// TwinCAT 3 PLC project PLC1
// ProgramVersion: 3.1.4024.12
// libraries:
//   Tc2_MC2, * (Beckhoff Automation GmbH)
//   Tc2_NC, * (Beckhoff Automation GmbH)
//   Tc2_Standard, * (Beckhoff Automation GmbH)
//   Tc2_System, * (Beckhoff Automation GmbH)
//   Tc3_MC2_AdvancedHoming, * (Beckhoff Automation GmbH)
//   Tc3_Module, * (Beckhoff Automation GmbH)
// project tree:
//   DUTs/ E_FT.TcTLEO, E_MoveState.TcDUT
//   GVLs/constants/ GVL_AlarmMessage.TcGVL, GVL_InitialSetting.TcGVL
//   GVLs/ GVL_HMI.TcGVL, GVL_IO.TcGVL, GVL_var.TcGVL
//   / PlcTask.TcTTO
//   POUs/BaseFuntion/ FB_CheckFeedback.TcPOU, FB_SetAlarm.TcPOU, FB_TransmitStatesToHMI.TcPOU
//   POUs/ FB_CasingVibratoryBowl1.TcPOU, FB_CorePress.TcPOU, FB_CoreSwaging.TcPOU, FB_CoreVibratoryBowl2.TcPOU, FB_Motor1.TcPOU, FB_OilPump.TcPOU, MAIN.TcPOU
// real-time tasks:
//   TASK PlcTask: cycle T#10ms, priority 20, ADS port 350
// motion (NC):
//   TASK NC-Task 1 SAF: cycle T#2ms, priority 4, ADS port 501
//   TASK NC-Task 1 SVB: cycle T#10ms, priority 8, ADS port 511
//   AXIS Axis 1 (id 1)
//     OtherSettings: AllowMotionCmdToSlave=true
//     encoder EncType=19
//       EncPara: MaxCount=#xffffffff
//     drive DrvType=16
//       DrvPara: MaxCount=#xffffffff, DriveControlDWord=#x00020000
//         Analog: TorqueSetpointScale=10, ScaleFactorActTorque=0.1
//         TimeComp: TaskDelayCycles=1
//     controller CtrType=1
//       CtrPara: PriorControlFactor=1
//         Observer: BandWidth=20
// I/O:
//   DEVICE Device 5 (EtherCAT), AmsNetId 169.254.43.171.6.1
//     Coupler (EK1100) [EK1100 EtherCAT Coupler (2A E-Bus)]
//       Slot1-DI (EL1809) [EL1809 16Ch. Dig. Input 24V, 3ms]
//       Slot2-DI (EL1809) [EL1809 16Ch. Dig. Input 24V, 3ms]
//       Slot3-DI (EL1809) [EL1809 16Ch. Dig. Input 24V, 3ms]
//       Slot4-AI (EL3072) [EL3072 2Ch. Ana. Input +/-10V, +/-20mA]
//       Slot5-DO (EL2809-0015) [EL2809-0015 16Ch. Dig. Output 24V DC, 0.35A, not short-circuit proof]
//       Slot6-DO (EL2809-0015) [EL2809-0015 16Ch. Dig. Output 24V DC, 0.35A, not short-circuit proof]
//       Slot7-DO (EL2809-0015) [EL2809-0015 16Ch. Dig. Output 24V DC, 0.35A, not short-circuit proof]
//       EndTerminal (EL9011) [EL9011 End Terminal]
//     Drive 9 (IHSS57/60-EC) [IHSS57/60-EC]
// variable links:
//   NC-Task 1 SAF/Axes/Axis 1 <-> Device 5 (EtherCAT)/Drive 9 (IHSS57/60-EC)
//     Drive/Inputs/In/nDcOutputTime <-> InfoData/DcOutputShift
//     Drive/Inputs/In/nState1 <-> TxPdoMapping/statusword
//     Drive/Inputs/In/nState2 <-> TxPdoMapping/statusword @bit 8
//     Drive/Inputs/In/nState4 @bit 1 <-> WcState/InputToggle
//     Drive/Inputs/In/nState4 <-> WcState/WcState
//     Drive/Inputs/In/nState5 <-> TxPdoMapping/op_mode_display
//     Drive/Outputs/Out/nCtrl1 <-> RxPdoMapping/controlword
//     Drive/Outputs/Out/nCtrl2 <-> RxPdoMapping/controlword @bit 8
//     Drive/Outputs/Out/nCtrl5 <-> RxPdoMapping/op_mode
//     Drive/Outputs/Out/nDataOut1 <-> RxPdoMapping/target_position
//     Enc/Inputs/In/nDataIn1 <-> TxPdoMapping/actual_position
//     Enc/Inputs/In/nDataIn3 <-> TxPdoMapping/Touch_probe_pos1_pos_value
//     Enc/Inputs/In/nDataIn5 <-> TxPdoMapping/Touch_probe_pos2_pos_value
//     Enc/Inputs/In/nDataIn4 <-> TxPdoMapping/Touch_probe_pos1_neg_value
//     Enc/Inputs/In/nDataIn6 <-> TxPdoMapping/Touch_probe_pos2_neg_value
//     Enc/Inputs/In/nDcInputTime <-> InfoData/DcInputShift
//     Enc/Inputs/In/nState4 @bit 1 <-> WcState/InputToggle
//     Enc/Inputs/In/nState4 <-> WcState/WcState
//     Enc/Inputs/In/nState5 <-> TxPdoMapping/Touch_probe_status
//     Enc/Inputs/In/nState6 <-> TxPdoMapping/Touch_probe_status @bit 8
//     Enc/Outputs/Out/nCtrl5 <-> RxPdoMapping/Touch_probe_function
//     Enc/Outputs/Out/nCtrl6 <-> RxPdoMapping/Touch_probe_function @bit 8
//   PLC1/PLC1 Instance <-> Device 5 (EtherCAT)/Coupler (EK1100)/Slot1-DI (EL1809)
//     PlcTask Inputs/GVL_IO.DI_24VDC_CB_OK <-> Channel 1/Input
//     PlcTask Inputs/GVL_IO.DI_CYL{1..6}_E <-> Channel {6..16 step 2}/Input  (6 links)
//     PlcTask Inputs/GVL_IO.DI_CYL{1..5}_R <-> Channel {7..15 step 2}/Input  (5 links)
//     PlcTask Inputs/GVL_IO.DI_ESR1 <-> Channel 2/Input
//     PlcTask Inputs/GVL_IO.DI_LS1 <-> Channel 4/Input
//     PlcTask Inputs/GVL_IO.DI_M1 <-> Channel 3/Input
//     PlcTask Inputs/GVL_IO.DI_TS1 <-> Channel 5/Input
//   PLC1/PLC1 Instance <-> Device 5 (EtherCAT)/Coupler (EK1100)/Slot2-DI (EL1809)
//     PlcTask Inputs/GVL_IO.DI_CYL6_R <-> Channel 1/Input
//     PlcTask Inputs/GVL_IO.DI_CYL7_R <-> Channel 3/Input
//     PlcTask Inputs/GVL_IO.DI_CYL7_E <-> Channel 2/Input
//     PlcTask Inputs/GVL_IO.DI_ECS <-> Channel 11/Input
//     PlcTask Inputs/GVL_IO.DI_EPD <-> Channel 12/Input
//     PlcTask Inputs/GVL_IO.DI_JLU <-> Channel 13/Input
//     PlcTask Inputs/GVL_IO.DI_PCYL1_E <-> Channel 7/Input
//     PlcTask Inputs/GVL_IO.DI_PCYL2_E <-> Channel 9/Input
//     PlcTask Inputs/GVL_IO.DI_PCYL1_R <-> Channel 8/Input
//     PlcTask Inputs/GVL_IO.DI_PCYL2_R <-> Channel 10/Input
//     PlcTask Inputs/GVL_IO.DI_PE1 <-> Channel 14/Input
//     PlcTask Inputs/GVL_IO.DI_PE2 <-> Channel 15/Input
//     PlcTask Inputs/GVL_IO.DI_PE3 <-> Channel 16/Input
//     PlcTask Inputs/GVL_IO.DI_PS1 <-> Channel 6/Input
//   PLC1/PLC1 Instance <-> Device 5 (EtherCAT)/Coupler (EK1100)/Slot3-DI (EL1809)
//     PlcTask Inputs/GVL_IO.DI_PE4 <-> Channel 1/Input
//     PlcTask Inputs/GVL_IO.DI_PE5 <-> Channel 2/Input
//     PlcTask Inputs/GVL_IO.DI_PE6 <-> Channel 3/Input
//   PLC1/PLC1 Instance <-> Device 5 (EtherCAT)/Coupler (EK1100)/Slot4-AI (EL3072)
//     PlcTask Inputs/GVL_IO.AI_PT1 <-> AI Standard Channel 1/Value
//     PlcTask Inputs/GVL_IO.AI_PT2 <-> AI Standard Channel 2/Value
//   PLC1/PLC1 Instance <-> Device 5 (EtherCAT)/Coupler (EK1100)/Slot5-DO (EL2809-0015)
//     PlcTask Outputs/GVL_IO.DO_CYL{1..6}_E <-> Channel {6..16 step 2}/Output  (6 links)
//     PlcTask Outputs/GVL_IO.DO_CYL{1..5}_R <-> Channel {7..15 step 2}/Output  (5 links)
//     PlcTask Outputs/GVL_IO.DO_M1 <-> Channel 1/Output
//     PlcTask Outputs/GVL_IO.DO_M2 <-> Channel 2/Output
//     PlcTask Outputs/GVL_IO.DO_SV1 <-> Channel 5/Output
//     PlcTask Outputs/GVL_IO.DO_VB1 <-> Channel 3/Output
//     PlcTask Outputs/GVL_IO.DO_VB2 <-> Channel 4/Output
//   PLC1/PLC1 Instance <-> Device 5 (EtherCAT)/Coupler (EK1100)/Slot6-DO (EL2809-0015)
//     PlcTask Outputs/GVL_IO.DO_CYL6_R <-> Channel 1/Output
//     PlcTask Outputs/GVL_IO.DO_CYL7_R <-> Channel 3/Output
//     PlcTask Outputs/GVL_IO.DO_CYL8_R <-> Channel 5/Output
//     PlcTask Outputs/GVL_IO.DO_CYL7_E <-> Channel 2/Output
//     PlcTask Outputs/GVL_IO.DO_CYL8_E <-> Channel 4/Output
//     PlcTask Outputs/GVL_IO.DO_LGreen <-> Channel 16/Output
//     PlcTask Outputs/GVL_IO.DO_PCYL1_E <-> Channel 6/Output
//     PlcTask Outputs/GVL_IO.DO_PCYL2_E <-> Channel 8/Output
//     PlcTask Outputs/GVL_IO.DO_PCYL3_E <-> Channel 10/Output
//     PlcTask Outputs/GVL_IO.DO_PCYL4_E <-> Channel 11/Output
//     PlcTask Outputs/GVL_IO.DO_PCYL5_E <-> Channel 12/Output
//     PlcTask Outputs/GVL_IO.DO_PCYL6_E <-> Channel 13/Output
//     PlcTask Outputs/GVL_IO.DO_PCYL1_R <-> Channel 7/Output
//     PlcTask Outputs/GVL_IO.DO_PCYL2_R <-> Channel 9/Output
//   PLC1/PLC1 Instance <-> Device 5 (EtherCAT)/Coupler (EK1100)/Slot7-DO (EL2809-0015)
//     PlcTask Outputs/GVL_IO.DO_LRed <-> Channel 1/Output
//   PLC1/PLC1 Instance <-> NC-Task 1 SAF/Axes/Axis 1
//     PlcTask Inputs/GVL_IO.AxisRef1.NcToPlc <-> Outputs/ToPlc
//     PlcTask Outputs/GVL_IO.AxisRef1.PlcToNc <-> Inputs/FromPlc

CONFIGURATION PLC1
    RESOURCE PLC ON TwinCAT3
        TASK PlcTask(INTERVAL := T#10ms, PRIORITY := 20);
        PROGRAM Main WITH PlcTask : Main;
    END_RESOURCE
END_CONFIGURATION

// ---- DUTs/E_FT.TcTLEO
{attribute 'qualified_only'}
{attribute 'strict'}
TYPE E_FT :
(
	PUMP,
	
	CYL1_E,
	CYL1_R,
	CYL2_E,
	CYL2_R,
	CYL3_E,
	CYL3_R,
	CYL4_E,
	CYL4_R,
	CYL5_E,
	CYL5_R,
	CYL6_E,
	CYL6_R,
	CYL7_E,
	CYL7_R,
	
	PCYL1_E,
	PCYL1_R,
	PCYL2_E,
	PCYL2_R
);
END_TYPE

// ---- DUTs/E_MoveState.TcDUT
{attribute 'qualified_only'}
{attribute 'strict'}
TYPE E_MoveState :
(
	init,
	enable,
	forward,
	backwards,
	backwards_slow,
	new_target_position,
	error,
	reset
);
END_TYPE

// ---- GVLs/constants/GVL_AlarmMessage.TcGVL
{attribute $27qualified_only$27}
VAR_GLOBAL CONSTANT
	DC : STRING := '24 DC Power Off!';
	ESR1 : STRING := 'Emergency Stop Relay 1 failed!';
	LS1 : STRING := 'Low Oil Level Sw failed!';
	TS1 : STRING := 'High Oil Temp Sw failed!';
	PS1 : STRING := 'Low Air Pressure Switch failed!';
	
	PUMP : STRING := 'Pump isn$27t started to run!';
	PUMP_OFF : STRING := 'Pump isn$27t stopped To run!';
	
	ECS : STRING := 'Operator interface Enable Core Swaging (Stayput Switch) failed!';
	
	CYL1_NOT_EXTENDED : STRING := 'Cylinder 1 isn$27t be extended!'; 
	CYL1_NOT_EXTENDED_OFF : STRING := 'Cylinder 1 isn$27t be de-extended!'; 
	CYL1_NOT_RETRACTED : STRING := 'Cylinder 1 isn$27t be retracted!'; 
	CYL1_NOT_RETRACTED_OFF : STRING := 'Cylinder 1 isn$27t be de-retracted!'; 
	CYL2_NOT_EXTENDED : STRING := 'Cylinder 2 isn$27t be extended!'; 
	CYL2_NOT_EXTENDED_OFF : STRING := 'Cylinder 2 isn$27t be de-extended!'; 
	CYL2_NOT_RETRACTED : STRING := 'Cylinder 2 isn$27t be retracted!';
	CYL2_NOT_RETRACTED_OFF : STRING := 'Cylinder 2 isn$27t be de-retracted!'; 
	CYL3_NOT_EXTENDED : STRING := 'Cylinder 3 isn$27t be extended!';  
	CYL3_NOT_EXTENDED_OFF : STRING := 'Cylinder 3 isn$27t be de-extended!'; 
	CYL3_NOT_RETRACTED : STRING := 'Cylinder 3 isn$27t be retracted!';
	CYL3_NOT_RETRACTED_OFF : STRING := 'Cylinder 3 isn$27t be de-retracted!'; 
	CYL4_NOT_EXTENDED : STRING := 'Cylinder 4 isn$27t be extended!';  
	CYL4_NOT_EXTENDED_OFF : STRING := 'Cylinder 4 isn$27t be de-extended!'; 
	CYL4_NOT_RETRACTED : STRING := 'Cylinder 4 isn$27t be retracted!';
	CYL4_NOT_RETRACTED_OFF : STRING := 'Cylinder 4 isn$27t be de-retracted!'; 
	CYL5_NOT_EXTENDED : STRING := 'Cylinder 5 isn$27t be extended!'; 
	CYL5_NOT_EXTENDED_OFF : STRING := 'Cylinder 5 isn$27t be de-extended!'; 
	CYL5_NOT_RETRACTED : STRING := 'Cylinder 5 isn$27t be retracted!'; 
	CYL5_NOT_RETRACTED_OFF : STRING := 'Cylinder 5 isn$27t be de-retracted!'; 
	CYL6_NOT_EXTENDED : STRING := 'Cylinder 6 isn$27t extended!'; 
	CYL6_NOT_EXTENDED_OFF : STRING := 'Cylinder 6 isn$27t de-extended!';
	CYL6_NOT_RETRACTED : STRING := 'Cylinder 6 isn$27t be retracted!';
	CYL6_NOT_RETRACTED_OFF : STRING := 'Cylinder 6 isn$27t be de-retracted!'; 
	CYL7_NOT_EXTENDED : STRING := 'Cylinder 7 isn$27t extended!'; 
	CYL7_NOT_EXTENDED_OFF : STRING := 'Cylinder 7 isn$27t de-extended!';
	CYL7_NOT_RETRACTED : STRING := 'Cylinder 7 isn$27t be retracted!';
	CYL7_NOT_RETRACTED_OFF : STRING := 'Cylinder 7 isn$27t be de-retracted!'; 
	
	PCYL1_NOT_EXTENDED : STRING := 'Pneumatic Cylinder 1 isn$27t be extended!';
	PCYL1_NOT_EXTENDED_OFF : STRING := 'Pneumatic Cylinder 1 isn$27t be de-extended!'; 
	PCYL1_NOT_RETRACTED : STRING := 'Pneumatic Cylinder 1 isn$27t be retracted!'; 
	PCYL1_NOT_RETRACTED_OFF : STRING := 'Pneumatic Cylinder 1 isn$27t be de-retracted!'; 
	PCYL2_NOT_EXTENDED : STRING := 'Pneumatic Cylinder 2 isn$27t be extended!'; 
	PCYL2_NOT_EXTENDED_OFF : STRING := 'Pneumatic Cylinder 2 isn$27t be de-extended!';
	PCYL2_NOT_RETRACTED : STRING := 'Pneumatic Cylinder 2 isn$27t be retracted!';
	PCYL2_NOT_RETRACTED_OFF : STRING := 'Pneumatic Cylinder 2 isn$27t be de-retracted!'; 
	
	// Vibratory
	PE1_FAIL : STRING := 'Vibratory Bowl 1 Product In Pos PE1 fail!';
	PE2_FAIL : STRING := 'Vibratory Bowl 1 Product Invert PE2 fail!';
	PE3_FAIL : STRING := 'Vibratory Bowl 2 Product In Pos PE3 fail!';
	PE4_FAIL : STRING := 'Vibratory Bowl 1 Product High Level PE4 fail!';	
	PE5_FAIL : STRING := 'Low Lead Spool!';
	
END_VAR

// ---- GVLs/constants/GVL_InitialSetting.TcGVL
{attribute 'qualified_only'}
VAR_GLOBAL CONSTANT
	PUMP_FeedbackCheckingTime : INT := 2000; // ms
	PUMP_RunningDelayTime : INT := 2000; // ms
	
	CYLINDER_FeedbackCheckingTime : INT := 3000; // ms
	
	PCYLINDER1EXTENDED_RunningTime: INT := 100;
	PCYLINDER1RETRACTED_RunningTime: INT := 100;
	PCYLINDER2EXTENDED_RunningTime: INT := 100;
	CYLINDER1EXTENDED_RunningTime: INT := 100;
	CYLINDER1RETRACTED_RunningTime: INT := 100;
	CYLINDER2EXTENDED_RunningTime: INT := 100;
	CYLINDER2RETRACTED_RunningTime: INT := 100;
	CYLINDER3EXTENDED_RunningTime: INT := 100;
	CYLINDER3RETRACTED_RunningTime: INT := 100;
	CYLINDER4EXTENDED_RunningTime: INT := 100;
	CYLINDER4RETRACTED_RunningTime: INT := 100;
	CYLINDER5EXTENDED_RunningDelayTime: INT := 250;
	CYLINDER5RETRACTED_RunningDelayTime: INT := 50;
	CYLINDER6RETRACTED_RunningDelayTime: INT := 50;
	CYLINDER6EXTENDED_RunningDelayTime: INT := 50;
	CYLINDER7RETRACTED_RunningDelayTime: INT := 50;
	CYLINDER7EXTENDED_RunningDelayTime: INT := 50;
	
	M3_RunningDelayTime : INT := 50;
	BOWL_RunningDelayTime : INT := 50;
	
	// for BOWL1
	PCYLINDER3EXTENDED_RunningTime: INT := 250;
	PE2_CheckingDelayTime: INT := 100;
	PE2_MaintainTime: INT := 10;
	PCYLINDER5EXTENDED_RunningTime: INT := 250;
	PCYLINDER4EXTENDED_RunningTime: INT := 150;
	PE4_MaintainTime: INT := 500;
	VB1_MaintainTime: INT := 50;
	
	// for BOWL2
	PCYLINDER6EXTENDED_RunningTime: INT := 250;
	PE6_MaintainTime: INT := 500;
	VB2_MaintainTime: INT := 50;
	
	PUMP_FAN_DelayTime : INT := 10000;
	PUMP_RestartingTime: INT := 3000;
	
	CASING_COUNT_FOR_STARTING : INT := 5;
	CORE_COUNT_FOR_STARTING : INT := 5;
END_VAR

// ---- GVLs/GVL_HMI.TcGVL
VAR_GLOBAL
	// Manual Control
	bManualControl : BOOL := FALSE;
		// motor1
	MC_M1_bSet : BOOL := FALSE;
	MC_M1_rPos : REAL := 0.0;
	MC_M1_rVel : REAL := 0.0;
	MC_M1_rAcc : REAL := 0.0;
	MC_M1_rDec : REAL := 0.0;	

	// safeties
	i_b24VDC_CB_OK : BOOL := FALSE;
	i_bESR1 : BOOL := FALSE;
	i_bLS1 : BOOL := FALSE;
	i_bTS1 : BOOL := FALSE;
	i_bPS1 : BOOL := FALSE;
	bSafeties :BOOL := TRUE;
	
	// signals from HMI
	i_nCmd_Reset : SINT := 0;	// reset Alarm; 0:NoAction, 1:Act, 2:AcceptToAct
	i_nCmd_ClearCount : SINT := 0;	// clear casing count and core count; 0:NoAction, 1:Act, 2:AcceptToAct
	i_nCmd_ResetSetting : SINT := 0;	// reset setting; 0:NoAction, 1:Act, 2:AcceptToAct
	i_nCmd_ResetAlarm : SINT := 0;	// reset Alarm; 0:NoAction, 1:Act, 2:AcceptToAct
	
		// settings
	i_nCoreSwagingMode: INT := 0;	// 0: Auto, 1: Manual
	i_nCasingCountForStarting : INT := GVL_InitialSetting.CASING_COUNT_FOR_STARTING;
	i_nCoreCountForStarting : INT := GVL_InitialSetting.CORE_COUNT_FOR_STARTING;
	i_nPumpFeedbackCheckingTime : INT := GVL_InitialSetting.PUMP_FeedbackCheckingTime; // ms
	i_nCylinderFeedbackCheckingTime : INT := GVL_InitialSetting.CYLINDER_FeedbackCheckingTime; // ms
	i_nPCylinder1ExtendedRunningTime : INT := GVL_InitialSetting.PCYLINDER1EXTENDED_RunningTime; // ms
	i_nCylinder3ExtendedRunningTime : INT := GVL_InitialSetting.CYLINDER3EXTENDED_RunningTime; // ms
	i_nCylinder1ExtendedRunningTime : INT := GVL_InitialSetting.CYLINDER1EXTENDED_RunningTime; // ms
	i_nPCylinder1RetractedRunningTime : INT := GVL_InitialSetting.PCYLINDER1RETRACTED_RunningTime; // ms
	i_nCylinder3RetractedRunningTime : INT := GVL_InitialSetting.CYLINDER3RETRACTED_RunningTime; // ms
	i_nCylinder1RetractedRunningTime : INT := GVL_InitialSetting.CYLINDER1RETRACTED_RunningTime; // ms
	i_nPCylinder2ExtendedRunningTime : INT := GVL_InitialSetting.PCYLINDER2EXTENDED_RunningTime; // ms
	i_nCylinder4ExtendedRunningTime : INT := GVL_InitialSetting.CYLINDER4EXTENDED_RunningTime; // ms
	i_nCylinder2ExtendedRunningTime : INT := GVL_InitialSetting.CYLINDER2EXTENDED_RunningTime; // ms
	i_nCylinder4RetractedRunningTime : INT := GVL_InitialSetting.CYLINDER4RETRACTED_RunningTime; // ms
	i_nCylinder2RetractedRunningTime : INT := GVL_InitialSetting.CYLINDER2RETRACTED_RunningTime; // ms
	i_nPCylinder3ExtendedRunningTime : INT := GVL_InitialSetting.PCYLINDER3EXTENDED_RunningTime; // ms
	i_nPCylinder5ExtendedRunningTime : INT := GVL_InitialSetting.PCYLINDER5EXTENDED_RunningTime; // ms
	i_nPCylinder4ExtendedRunningTime : INT := GVL_InitialSetting.PCYLINDER4EXTENDED_RunningTime; // ms
	i_nPE4MaintainTime : INT := GVL_InitialSetting.PE4_MaintainTime; // ms
	i_nPCylinder6ExtendedRunningTime : INT := GVL_InitialSetting.PCYLINDER6EXTENDED_RunningTime; // ms
	i_nPE6MaintainTime : INT := GVL_InitialSetting.PE6_MaintainTime; // ms
	
	// output
	i_bVB1 : BOOL := FALSE;
	i_bVB2 : BOOL := FALSE;
	i_bCyl1E : BOOL := FALSE;
	i_bCyl1R : BOOL := FALSE;
	i_bCyl2E : BOOL := FALSE;
	i_bCyl2R : BOOL := FALSE;
	i_bCyl3E : BOOL := FALSE;
	i_bCyl3R : BOOL := FALSE;
	i_bCyl4E : BOOL := FALSE;
	i_bCyl4R : BOOL := FALSE;
	i_bCyl5E : BOOL := FALSE;
	i_bCyl5R : BOOL := FALSE;
	i_bCyl6E : BOOL := FALSE;
	i_bCyl6R : BOOL := FALSE;
	i_bCyl7E : BOOL := FALSE;
	i_bCyl7R : BOOL := FALSE;
	i_bCyl8E : BOOL := FALSE;
	i_bCyl8R : BOOL := FALSE;
	
	// core swagging
	i_bECS : BOOL := FALSE;
	i_bEPD : BOOL := FALSE;
	i_bJLU : BOOL := FALSE;
	
	// pump
	i_nPumpState : SINT := 0; // 0: InitialState, -1:Faulted, 1: StartingToRun, 2:Running, 3:Stopping, 4:Stopped
	// cylinders
	i_nCylinder1State : SINT := 0; // 0: InitialState, -3: FaultedWhileRetracting, -1: FaultedWhileExtending, 1: Extending, 2:Extended, 3:Retracting, 4: Retracted
	i_nCylinder2State : SINT := 0; // 0: InitialState, -3: FaultedWhileRetracting, -1: FaultedWhileExtending, 1: Extending, 2:Extended, 3:Retracting, 4: Retracted
	i_nCylinder3State : SINT := 0; // 0: InitialState, -3: FaultedWhileRetracting, -1: FaultedWhileExtending, 1: Extending, 2:Extended, 3:Retracting, 4: Retracted
	i_nCylinder4State : SINT := 0; // 0: InitialState, -3: FaultedWhileRetracting, -1: FaultedWhileExtending, 1: Extending, 2:Extended, 3:Retracting, 4: Retracted
	i_nCylinder5State : SINT := 0; // 0: InitialState, -3: FaultedWhileRetracting, -1: FaultedWhileExtending, 1: Extending, 2:Extended, 3:Retracting, 4: Retracted
	i_nCylinder6State : SINT := 0; // 0: InitialState, -3: FaultedWhileRetracting, -1: FaultedWhileExtending, 1: Extending, 2:Extended, 3:Retracting, 4: Retracted
	i_nCylinder7State : SINT := 0; // 0: InitialState, -3: FaultedWhileRetracting, -1: FaultedWhileExtending, 1: Extending, 2:Extended, 3:Retracting, 4: Retracted
	i_nCylinder8State : SINT := 0; // 0: InitialState, -3: FaultedWhileRetracting, -1: FaultedWhileExtending, 1: Extending, 2:Extended, 3:Retracting, 4: Retracted
	i_nPCylinder1State : SINT := 0; // 0: InitialState, -3: FaultedWhileRetracting, -1: FaultedWhileExtending, 1: Extending, 2:Extended, 3:Retracting, 4: Retracted
	i_nPCylinder2State : SINT := 0; // 0: InitialState, -3: FaultedWhileRetracting, -1: FaultedWhileExtending, 1: Extending, 2:Extended, 3:Retracting, 4: Retracted
	
	// Vibratory
	i_bPE1 : BOOL := FALSE;
	i_bPE2 : BOOL := FALSE;
	i_bPE3 : BOOL := FALSE;
	i_bPE4 : BOOL := FALSE;
	i_bPE5 : BOOL := FALSE;
	
	// Analog Value
	i_rPT1 : REAL := 1.0;
	i_rPT2 : REAL := 1.0;
	
	// working count
	nProductCount : INT := 0;
	nCasingCount: INT := 0;
	nCoreCount: INT := 0;
	
	// alram message
	o_bAlarmActive: BOOL := FALSE;
	o_sAlarmMessage: STRING := '';
	
	// active alarm
		// Safeties
	nAlarmSafeties : SINT := 0;		// 0: Init, 1: OK, -1: Fail
	nAlarmS_24DC : SINT :=0;	// 0: Init, 1: OK, -1: Fail
	nAlarmS_ESR1 : SINT :=0;	// 0: Init, 1: OK, -1: Fail
	nAlarmS_LS1 : SINT :=0;	// 0: Init, 1: OK, -1: Fail
	nAlarmS_TS1 : SINT :=0;	// 0: Init, 1: OK, -1: Fail
	nAlarmS_PS1 : SINT :=0;	// 0: Init, 1: OK, -1: Fail
		// core swagging
	nAlarmCS_10_ECS : SINT := 0;	// 0: Init, 1: On, -1: Off
	nAlarmCS_10_Pump : SINT :=0;	// 0: Init, 1: OK, -1: Fail
	nAlarmCS_20_HC6E : SINT :=0;	// 0: Init, 1: OK, -1: Fail
	nAlarmCS_21_HC5R : SINT :=0;	// 0: Init, 1: OK, -1: Fail
	nAlarmCS_30_HC7R : SINT :=0;	// 0: Init, 1: OK, -1: Fail
	nAlarmCS_40_PE5 : SINT := 0;	// 0: Init, 1: On, -1: Off
	nAlarmCS_50_HC7E : SINT :=0;	// 0: Init, 1: OK, -1: Fail
	nAlarmCS_60_HC6R : SINT :=0;	// 0: Init, 1: OK, -1: Fail
	nAlarmCS_70_HC5E : SINT :=0;	// 0: Init, 1: OK, -1: Fail
	nAlarmCS_80_HC5R : SINT :=0;	// 0: Init, 1: OK, -1: Fail
		// core pressing
	nAlarmCP_10_EPD : SINT := 0;	// 0: Init, 1: On, -1: Off
	nAlarmCP_10_Pump : SINT :=0;	// 0: Init, 1: OK, -1: Fail
	nAlarmCP_10_HC1R : SINT :=0;
	nAlarmCP_20_PC1E : SINT :=0;
	nAlarmCP_10_PC1R : SINT :=0;
	nAlarmCP_10_HC3R : SINT :=0;
	nAlarmCP_50_HC1R : SINT :=0;
	nAlarmCP_10_PC2E : SINT :=0;
	nAlarmCP_10_HC4E : SINT :=0;
	nAlarmCP_10_HC2E : SINT :=0;
	nAlarmCP_10_HC4R : SINT :=0;
	nAlarmCP_10_HC2R : SINT :=0;
END_VAR

// ---- GVLs/GVL_IO.TcGVL
{attribute 'qualified_only'}
VAR_GLOBAL
	AxisRef1 : AXIS_REF;

	DI_24VDC_CB_OK 	AT %I*: BOOL := FALSE;
	DI_ESR1 		AT %I*: BOOL := FALSE;
	DI_M1 			AT %I*: BOOL := FALSE;
	DI_LS1	 		AT %I*: BOOL := FALSE;
	DI_TS1 			AT %I*: BOOL := FALSE;
	DI_CYL1_E 		AT %I*: BOOL := FALSE;
	DI_CYL1_R 		AT %I*: BOOL := FALSE;
	DI_CYL2_E 		AT %I*: BOOL := FALSE;
	DI_CYL2_R 		AT %I*: BOOL := FALSE;
	DI_CYL3_E 		AT %I*: BOOL := FALSE;
	DI_CYL3_R 		AT %I*: BOOL := FALSE;
	DI_CYL4_E 		AT %I*: BOOL := FALSE;
	DI_CYL4_R 		AT %I*: BOOL := FALSE;
	DI_CYL5_E 		AT %I*: BOOL := FALSE;
	DI_CYL5_R 		AT %I*: BOOL := FALSE;
	DI_CYL6_E 		AT %I*: BOOL := FALSE;
	DI_CYL6_R 		AT %I*: BOOL := FALSE;
	DI_CYL7_E 		AT %I*: BOOL := FALSE;
	DI_CYL7_R 		AT %I*: BOOL := FALSE;
	DI_PS1			AT %I*: BOOL := FALSE;
	DI_PCYL1_E		AT %I*: BOOL := FALSE;
	DI_PCYL1_R		AT %I*: BOOL := FALSE;
	DI_PCYL2_E		AT %I*: BOOL := FALSE;
	DI_PCYL2_R		AT %I*: BOOL := FALSE;
	DI_ECS			AT %I*: BOOL := FALSE;
	DI_EPD			AT %I*: BOOL := FALSE;
	DI_JLU			AT %I*: BOOL := FALSE;

	DI_PE1			AT %I*: BOOL := FALSE;
	DI_PE2			AT %I*: BOOL := FALSE;
	DI_PE3			AT %I*: BOOL := FALSE;
	DI_PE4			AT %I*: BOOL := FALSE;
	DI_PE5			AT %I*: BOOL := FALSE;
	DI_PE6			AT %I*: BOOL := FALSE;
	
	AI_PT1			AT %I*: INT := 1;
	AI_PT2			AT %I*: INT := 1;

	DO_M1			AT %Q*: BOOL;
	DO_M2			AT %Q*: BOOL;
	DO_VB1			AT %Q*: BOOL;
	DO_VB2			AT %Q*: BOOL;
	DO_SV1			AT %Q*: BOOL;
	DO_CYL1_E		AT %Q*: BOOL;
	DO_CYL1_R		AT %Q*: BOOL;
	DO_CYL2_E		AT %Q*: BOOL;
	DO_CYL2_R		AT %Q*: BOOL;
	DO_CYL3_E		AT %Q*: BOOL;
	DO_CYL3_R		AT %Q*: BOOL;
	DO_CYL4_E		AT %Q*: BOOL;
	DO_CYL4_R		AT %Q*: BOOL;
	DO_CYL5_E		AT %Q*: BOOL;
	DO_CYL5_R		AT %Q*: BOOL;
	DO_CYL6_E		AT %Q*: BOOL;
	DO_CYL6_R		AT %Q*: BOOL;
	DO_CYL7_E		AT %Q*: BOOL;
	DO_CYL7_R		AT %Q*: BOOL;
	DO_CYL8_E		AT %Q*: BOOL;
	DO_CYL8_R		AT %Q*: BOOL;
	DO_PCYL1_E		AT %Q*: BOOL;
	DO_PCYL1_R		AT %Q*: BOOL;
	DO_PCYL2_E		AT %Q*: BOOL;
	DO_PCYL2_R		AT %Q*: BOOL;
	DO_PCYL3_E		AT %Q*: BOOL;
	DO_PCYL4_E		AT %Q*: BOOL;
	DO_PCYL5_E		AT %Q*: BOOL;
	DO_PCYL6_E		AT %Q*: BOOL;
	DO_LGreen		AT %Q*: BOOL;
	DO_LRed			AT %Q*: BOOL;
END_VAR

// ---- GVLs/GVL_var.TcGVL
{attribute 'qualified_only'}
VAR_GLOBAL
	fMotor1: FB_Motor1;
	Motor1_bNew: BOOL := FALSE;
	Motor1_rPos: REAL := 0;
	Motor1_rVel: REAL := 0;
	Motor1_rAcc: REAL := 0;
	Motor1_rDec: REAL := 0;
END_VAR

// ---- POUs/MAIN.TcPOU
PROGRAM Main
VAR
	fSetAlarm : FB_SetAlarm;
	fCoreSwaging: FB_CoreSwaging;
    fOilPump: FB_OilPump;
    fCorePress: FB_CorePress;
    fCasingVibratoryBowl1: FB_CasingVibratoryBowl1;
    fCoreVibratoryBowl2: FB_CoreVibratoryBowl2;
	fTransmitStatesToHMI: FB_TransmitStatesToHMI;
	
	pAlarm : POINTER TO SINT;
	i : INT;
END_VAR

GVL_HMI.bSafeties := GVL_IO.DI_24VDC_CB_OK AND GVL_IO.DI_ESR1 AND GVL_IO.DI_LS1 AND GVL_IO.DI_TS1 AND GVL_IO.DI_PS1;

// accept commands
IF GVL_HMI.i_nCmd_ClearCount = 1 THEN GVL_HMI.i_nCmd_ClearCount := 2; END_IF
IF GVL_HMI.i_nCmd_Reset = 1 THEN GVL_HMI.i_nCmd_Reset := 2; END_IF
IF GVL_HMI.i_nCmd_ResetSetting = 1 THEN GVL_HMI.i_nCmd_ResetSetting := 2; END_IF
IF GVL_HMI.i_nCmd_ResetAlarm = 1 THEN GVL_HMI.i_nCmd_ResetAlarm := 2; END_IF

// reset alarm
IF GVL_HMI.i_nCmd_ResetAlarm = 2 THEN
	GVL_HMI.o_bAlarmActive := FALSE;
	pAlarm := ADR(GVL_HMI.nAlarmSafeties);
	FOR i := 0 TO 20 DO
		pAlarm[i] := 0;
	END_FOR
END_IF

// reset
IF GVL_HMI.i_nCmd_Reset = 2 THEN
	GVL_HMI.o_bAlarmActive := FALSE;
END_IF

// reset setting
IF GVL_HMI.i_nCmd_ResetSetting = 2 THEN
	GVL_HMI.i_nCoreSwagingMode:= 0;	// 0: Auto, 1: Manual
	GVL_HMI.i_nCasingCountForStarting := GVL_InitialSetting.CASING_COUNT_FOR_STARTING;
	GVL_HMI.i_nCoreCountForStarting := GVL_InitialSetting.CORE_COUNT_FOR_STARTING;
	GVL_HMI.i_nPumpFeedbackCheckingTime := GVL_InitialSetting.PUMP_FeedbackCheckingTime; // ms
	GVL_HMI.i_nCylinderFeedbackCheckingTime := GVL_InitialSetting.CYLINDER_FeedbackCheckingTime; // ms
	GVL_HMI.i_nPCylinder1ExtendedRunningTime := GVL_InitialSetting.PCYLINDER1EXTENDED_RunningTime; // ms
	GVL_HMI.i_nCylinder3ExtendedRunningTime := GVL_InitialSetting.CYLINDER3EXTENDED_RunningTime; // ms
	GVL_HMI.i_nCylinder1ExtendedRunningTime := GVL_InitialSetting.CYLINDER1EXTENDED_RunningTime; // ms
	GVL_HMI.i_nPCylinder1RetractedRunningTime := GVL_InitialSetting.PCYLINDER1RETRACTED_RunningTime; // ms
	GVL_HMI.i_nCylinder3RetractedRunningTime := GVL_InitialSetting.CYLINDER3RETRACTED_RunningTime; // ms
	GVL_HMI.i_nCylinder1RetractedRunningTime := GVL_InitialSetting.CYLINDER1RETRACTED_RunningTime; // ms
	GVL_HMI.i_nPCylinder2ExtendedRunningTime := GVL_InitialSetting.PCYLINDER2EXTENDED_RunningTime; // ms
	GVL_HMI.i_nCylinder4ExtendedRunningTime := GVL_InitialSetting.CYLINDER4EXTENDED_RunningTime; // ms
	GVL_HMI.i_nCylinder2ExtendedRunningTime := GVL_InitialSetting.CYLINDER2EXTENDED_RunningTime; // ms
	GVL_HMI.i_nCylinder4RetractedRunningTime := GVL_InitialSetting.CYLINDER4RETRACTED_RunningTime; // ms
	GVL_HMI.i_nCylinder2RetractedRunningTime := GVL_InitialSetting.CYLINDER2RETRACTED_RunningTime; // ms
	GVL_HMI.i_nPCylinder3ExtendedRunningTime := GVL_InitialSetting.PCYLINDER3EXTENDED_RunningTime; // ms
	GVL_HMI.i_nPCylinder5ExtendedRunningTime := GVL_InitialSetting.PCYLINDER5EXTENDED_RunningTime; // ms
	GVL_HMI.i_nPCylinder4ExtendedRunningTime := GVL_InitialSetting.PCYLINDER4EXTENDED_RunningTime; // ms
	GVL_HMI.i_nPE4MaintainTime := GVL_InitialSetting.PE4_MaintainTime; // ms
	GVL_HMI.i_nPCylinder6ExtendedRunningTime := GVL_InitialSetting.PCYLINDER6EXTENDED_RunningTime; // ms
	GVL_HMI.i_nPE6MaintainTime := GVL_InitialSetting.PE6_MaintainTime; // ms
END_IF

IF NOT GVL_HMI.o_bAlarmActive THEN
	IF GVL_IO.DI_24VDC_CB_OK THEN
		GVL_HMI.nAlarmS_24DC := 1;
	ELSE
		GVL_HMI.nAlarmS_24DC := -1;
		GVL_HMI.nAlarmSafeties := -1;
		fSetAlarm( sMsg := GVL_AlarmMessage.DC );
	END_IF
END_IF
IF NOT GVL_HMI.o_bAlarmActive THEN
	IF GVL_IO.DI_ESR1 THEN
		GVL_HMI.nAlarmS_ESR1 := 1;
	ELSE
		GVL_HMI.nAlarmS_ESR1 := -1;
		GVL_HMI.nAlarmSafeties := -1;
		fSetAlarm( sMsg := GVL_AlarmMessage.ESR1 );
	END_IF
END_IF
IF NOT GVL_HMI.o_bAlarmActive THEN
	IF GVL_IO.DI_LS1 THEN
		GVL_HMI.nAlarmS_LS1 := 1;
	ELSE
		GVL_HMI.nAlarmS_LS1 := -1;
		GVL_HMI.nAlarmSafeties := -1;
		fSetAlarm( sMsg := GVL_AlarmMessage.LS1 );
	END_IF
END_IF
IF NOT GVL_HMI.o_bAlarmActive THEN
	IF GVL_IO.DI_TS1 THEN
		GVL_HMI.nAlarmS_TS1 := 1;
	ELSE
		GVL_HMI.nAlarmS_TS1 := -1;
		GVL_HMI.nAlarmSafeties := -1;
		fSetAlarm( sMsg := GVL_AlarmMessage.TS1 );
	END_IF
END_IF
IF NOT GVL_HMI.o_bAlarmActive THEN
	IF GVL_IO.DI_PS1 THEN
		GVL_HMI.nAlarmS_PS1 := 1;
	ELSE
		GVL_HMI.nAlarmS_PS1 := -1;
		GVL_HMI.nAlarmSafeties := -1;
		fSetAlarm( sMsg := GVL_AlarmMessage.PS1 );
	END_IF
END_IF

IF GVL_HMI.bManualControl THEN
	IF GVL_HMI.MC_M1_bSet THEN
		GVL_HMI.MC_M1_bSet := FALSE;
		GVL_Var.Motor1_bNew := TRUE;
		GVL_Var.Motor1_rPos := GVL_HMI.MC_M1_rPos;
		GVL_Var.Motor1_rVel := GVL_HMI.MC_M1_rVel;
		GVL_Var.Motor1_rAcc := GVL_HMI.MC_M1_rAcc;
		GVL_Var.Motor1_rDec := GVL_HMI.MC_M1_rDec;
	ELSE
		GVL_Var.Motor1_bNew := FALSE;
	END_IF
ELSE
	IF NOT GVL_HMI.o_bAlarmActive THEN
		fCoreSwaging();
		fOilPump();
		fCorePress();
		fCasingVibratoryBowl1();
		fCoreVibratoryBowl2();
	END_IF
END_IF

GVL_Var.fMotor1( new:=GVL_Var.Motor1_bNew, pos:=GVL_Var.Motor1_rPos, vel:=GVL_Var.Motor1_rVel, acc:=GVL_Var.Motor1_rAcc, dec:=GVL_Var.Motor1_rDec );

fTransmitStatesToHMI();

// release commands
IF GVL_HMI.i_nCmd_ClearCount = 2 THEN GVL_HMI.i_nCmd_ClearCount := 0; END_IF
IF GVL_HMI.i_nCmd_Reset = 2 THEN GVL_HMI.i_nCmd_Reset := 0; END_IF
IF GVL_HMI.i_nCmd_ResetSetting = 2 THEN GVL_HMI.i_nCmd_ResetSetting := 0; END_IF
IF GVL_HMI.i_nCmd_ResetAlarm = 2 THEN GVL_HMI.i_nCmd_ResetAlarm := 0; END_IF

END_PROGRAM

// ---- POUs/BaseFuntion/FB_SetAlarm.TcPOU
FUNCTION_BLOCK FB_SetAlarm
VAR_INPUT
	sMSg : STRING := '';
END_VAR
VAR_OUTPUT
END_VAR
VAR
END_VAR

GVL_HMI.o_bAlarmActive := TRUE;
GVL_HMI.o_sAlarmMessage := sMSg;

END_FUNCTION_BLOCK

// ---- POUs/FB_CoreSwaging.TcPOU
FUNCTION_BLOCK FB_CoreSwaging
VAR_INPUT
END_VAR
VAR_OUTPUT
END_VAR
VAR
    iState : INT := 0;
	FeedbackTimer : TON;
    DelayTimer : TON;
	fSetAlarm : FB_SetAlarm;
	fCheckFeedback : FB_CheckFeedback;
END_VAR

CASE iState OF
	0: (* Idle/Off, DI_ECS=FALSE *)
		(* Manual Mode Handling *)
		IF GVL_HMI.i_nCoreSwagingMode = 1 THEN
			IF GVL_IO.DI_JLU THEN (* Jog switch pressed *)
				(* Motor M3 runs infinitely while switch is pressed *)
				iState := 10;
			END_IF
		ELSE
			iState := 10;
		END_IF
		
	10: (* check safety conditions *)
		IF GVL_HMI.bSafeties THEN (* Safeties OK*)
			IF GVL_IO.DI_ECS THEN (* Enable Switch On *)
				GVL_IO.DO_M1 := TRUE; (* Start Oil Pump *)
				CheckFeedback(E_FT.PUMP);
				IF GVL_IO.DI_M1 THEN
					DelayAndAdvance(GVL_InitialSetting.PUMP_RunningDelayTime, iState+10);
					GVL_HMI.nAlarmCS_10_Pump := 1;
				ELSIF FeedbackTimer.Q THEN
					GVL_HMI.nAlarmCS_10_Pump := -1;
				END_IF
				GVL_HMI.nAlarmCS_10_ECS := 1;
			ELSE
				GVL_HMI.nAlarmCS_10_ECS := -1;
				fSetAlarm( sMsg := GVL_AlarmMessage.ECS );
			END_IF
        END_IF
		
    20: (* Ensure CYL6 is Extended *)
        IF NOT GVL_IO.DI_CYL6_E THEN
			GVL_IO.DO_SV1 := TRUE;	// Power Pack Hydraulic Pressure Relief Valve
            GVL_IO.DO_CYL6_E := TRUE;
			CheckFeedback(E_FT.CYL6_E);
			IF FeedbackTimer.Q THEN GVL_HMI.nAlarmCS_20_HC6E := -1; END_IF
        ELSE
			GVL_HMI.nAlarmCS_20_HC6E := 1;
			DelayAndAdvance(GVL_InitialSetting.CYLINDER6EXTENDED_RunningDelayTime, iState+1);
        END_IF
	21: (* Ensure CYL5 is Retracted *)
    	IF NOT GVL_IO.DI_CYL5_R THEN
			GVL_IO.DO_CYL5_R := TRUE;
			CheckFeedback(E_FT.CYL5_R);
			IF FeedbackTimer.Q THEN GVL_HMI.nAlarmCS_21_HC5R := -1; END_IF
		ELSE
			GVL_HMI.nAlarmCS_21_HC5R := 1;
			iState := (iState + 10) / 10 * 10;
		END_IF
		
    30: (* Ensure CYL7 is Retracted *)
        IF NOT GVL_IO.DI_CYL7_R THEN
            GVL_IO.DO_CYL7_R := TRUE;
			CheckFeedback(E_FT.CYL7_R);
			IF FeedbackTimer.Q THEN GVL_HMI.nAlarmCS_30_HC7R := -1; END_IF
        ELSE
			GVL_HMI.nAlarmCS_30_HC7R := 1;
			DelayAndAdvance(GVL_InitialSetting.CYLINDER7RETRACTED_RunningDelayTime, iState+10);
        END_IF
    
    40: (* Low Lead Spool Check *)
        IF NOT GVL_IO.DI_PE5 THEN
			fSetAlarm( sMsg := GVL_AlarmMessage.PE5_FAIL );
			GVL_HMI.nAlarmCS_40_PE5 := -1;
        ELSE
			GVL_HMI.nAlarmCS_40_PE5 := 1;
			IF GVL_IO.DI_CYL4_R THEN
				(* index M3 *)
				
				iState := iState + 1;
			END_IF
        END_IF
	41: 
		DelayAndAdvance(GVL_InitialSetting.M3_RunningDelayTime, (iState + 10) / 10 * 10);
    
    50: (* Extend CYL7 *)
        IF NOT GVL_IO.DI_CYL7_E THEN
			GVL_IO.DO_CYL7_E := TRUE;
			CheckFeedback(E_FT.CYL7_E);
			IF FeedbackTimer.Q THEN GVL_HMI.nAlarmCS_50_HC7E := -1; END_IF
        ELSE
			GVL_HMI.nAlarmCS_50_HC7E := 1;
			DelayAndAdvance(GVL_InitialSetting.CYLINDER7EXTENDED_RunningDelayTime, iState + 10);
        END_IF
    
    60: (* Retract CYL6 *)
        IF NOT GVL_IO.DI_CYL6_R THEN
			GVL_IO.DO_CYL6_R := TRUE;
			CheckFeedback(E_FT.CYL6_R);
			IF FeedbackTimer.Q THEN GVL_HMI.nAlarmCS_60_HC6R := -1; END_IF
        ELSE
			GVL_HMI.nAlarmCS_60_HC6R := 1;
			DelayAndAdvance(GVL_InitialSetting.CYLINDER6RETRACTED_RunningDelayTime, iState + 10);
        END_IF
    
    70: (* Extend CYL5 *)
        IF NOT GVL_IO.DI_CYL5_E THEN
			GVL_IO.DO_CYL5_E := TRUE;
			CheckFeedback(E_FT.CYL5_E);
			IF FeedbackTimer.Q THEN GVL_HMI.nAlarmCS_70_HC5E := -1; END_IF
        ELSE
			GVL_HMI.nAlarmCS_70_HC5E := 1;
			DelayAndAdvance(GVL_InitialSetting.CYLINDER5EXTENDED_RunningDelayTime, iState + 10);
        END_IF
    
    80: (* Retract CYL5 *)
        IF NOT GVL_IO.DI_CYL5_R THEN
			GVL_IO.DO_CYL5_R := TRUE;
			CheckFeedback(E_FT.CYL5_R);
			IF FeedbackTimer.Q THEN GVL_HMI.nAlarmCS_80_HC5R := -1; END_IF
		ELSE
			GVL_HMI.nAlarmCS_80_HC5R := 1;
			DelayAndAdvance(GVL_InitialSetting.CYLINDER5RETRACTED_RunningDelayTime, iState + 10);
        END_IF
		
	90: (* Future Step *)
		iState := 20;
END_CASE

METHOD CheckFeedback : BOOL
VAR_INPUT
	t : E_FT;
END_VAR
VAR_OUTPUT
	o_nResult : INT := 0;	// -1: fail, 0: checking, 1: success 
END_VAR
fCheckFeedback(t:=t, FeedbackTimer:=FeedbackTimer);
o_nResult := fCheckFeedback.o_nResult;
END_METHOD

METHOD DelayAndAdvance : BOOL
VAR_INPUT
	i_nDelayTime: INT;	// ms
	i_nNextState: INT;
END_VAR

VAR
END_VAR
IF NOT DelayTimer.IN THEN
    DelayTimer(IN := TRUE, PT := INT_TO_TIME(i_nDelayTime));
ELSE
    IF DelayTimer.Q THEN 
        iState := i_nNextState; 
    END_IF
END_IF
END_METHOD

END_FUNCTION_BLOCK

// ---- POUs/BaseFuntion/FB_CheckFeedback.TcPOU
FUNCTION_BLOCK FB_CheckFeedback
VAR_INPUT
	t : E_FT;
	bRising: BOOL := TRUE;
END_VAR
VAR_IN_OUT
	FeedbackTimer : TON;
END_VAR
VAR_OUTPUT
	o_nResult : INT := 0;	// -1: fail, 0: checking, 1: success 
END_VAR
VAR
	bFeedback : BOOL;
	nCheckingTime: INT;
	sAlarmMessage: STRING;
	sMsg: INT;
	fSetAlarm : FB_SetAlarm;
END_VAR

CASE t OF
	E_FT.PUMP:
		bFeedback := GVL_IO.DI_M1;
		IF bRising THEN GVL_HMI.i_nPumpState := 1; ELSE GVL_HMI.i_nPumpState := 3; END_IF
	E_FT.CYL1_E:
		bFeedback := GVL_IO.DI_CYL1_E;
		IF bRising THEN GVL_HMI.i_nCylinder1State := 1; ELSE GVL_HMI.i_nCylinder1State := 0; END_IF
	E_FT.CYL1_R:
		bFeedback := GVL_IO.DI_CYL1_R;
		IF bRising THEN GVL_HMI.i_nCylinder1State := 3; ELSE GVL_HMI.i_nCylinder1State := 0; END_IF
	E_FT.CYL2_E:
		bFeedback := GVL_IO.DI_CYL2_E;
		IF bRising THEN GVL_HMI.i_nCylinder2State := 1; ELSE GVL_HMI.i_nCylinder2State := 0; END_IF
	E_FT.CYL2_R:
		bFeedback := GVL_IO.DI_CYL2_R;
		IF bRising THEN GVL_HMI.i_nCylinder2State := 3; ELSE GVL_HMI.i_nCylinder2State := 0; END_IF
	E_FT.CYL3_E:
		bFeedback := GVL_IO.DI_CYL3_E;
		IF bRising THEN GVL_HMI.i_nCylinder3State := 1; ELSE GVL_HMI.i_nCylinder1State := 0; END_IF
	E_FT.CYL3_R:
		bFeedback := GVL_IO.DI_CYL3_R;
		IF bRising THEN GVL_HMI.i_nCylinder3State := 3; ELSE GVL_HMI.i_nCylinder3State := 0; END_IF
	E_FT.CYL4_E:
		bFeedback := GVL_IO.DI_CYL4_E;
		IF bRising THEN GVL_HMI.i_nCylinder4State := 1; ELSE GVL_HMI.i_nCylinder4State := 0; END_IF
	E_FT.CYL4_R:
		bFeedback := GVL_IO.DI_CYL4_R;
		IF bRising THEN GVL_HMI.i_nCylinder4State := 3; ELSE GVL_HMI.i_nCylinder4State := 0; END_IF
	E_FT.CYL5_E:
		bFeedback := GVL_IO.DI_CYL5_E;
		IF bRising THEN GVL_HMI.i_nCylinder5State := 1; ELSE GVL_HMI.i_nCylinder5State := 0; END_IF
	E_FT.CYL5_R:
		bFeedback := GVL_IO.DI_CYL5_R;
		IF bRising THEN GVL_HMI.i_nCylinder5State := 3; ELSE GVL_HMI.i_nCylinder5State := 0; END_IF
	E_FT.CYL6_E:
		bFeedback := GVL_IO.DI_CYL6_E;
		IF bRising THEN GVL_HMI.i_nCylinder6State := 1; ELSE GVL_HMI.i_nCylinder6State := 0; END_IF
	E_FT.CYL6_R:
		bFeedback := GVL_IO.DI_CYL6_R;
		IF bRising THEN GVL_HMI.i_nCylinder6State := 3; ELSE GVL_HMI.i_nCylinder6State := 0; END_IF
	E_FT.CYL7_E:
		bFeedback := GVL_IO.DI_CYL7_E;
		IF bRising THEN GVL_HMI.i_nCylinder7State := 1; ELSE GVL_HMI.i_nCylinder7State := 0; END_IF
	E_FT.CYL7_R:
		bFeedback := GVL_IO.DI_CYL7_R;
		IF bRising THEN GVL_HMI.i_nCylinder7State := 3; ELSE GVL_HMI.i_nCylinder7State := 0; END_IF
	E_FT.PCYL1_E:
		bFeedback := GVL_IO.DI_PCYL1_E;
		IF bRising THEN GVL_HMI.i_nPCylinder1State := 1; ELSE GVL_HMI.i_nPCylinder1State := 0; END_IF
	E_FT.PCYL1_R:
		bFeedback := GVL_IO.DI_PCYL1_R;
		IF bRising THEN GVL_HMI.i_nPCylinder1State := 3; ELSE GVL_HMI.i_nPCylinder1State := 0; END_IF
	E_FT.PCYL2_E:
		bFeedback := GVL_IO.DI_PCYL2_E;
		IF bRising THEN GVL_HMI.i_nPCylinder2State := 1; ELSE GVL_HMI.i_nPCylinder2State := 0; END_IF
	E_FT.PCYL2_R:
		bFeedback := GVL_IO.DI_PCYL2_R;
		IF bRising THEN GVL_HMI.i_nPCylinder2State := 3; ELSE GVL_HMI.i_nPCylinder2State := 0; END_IF
END_CASE
IF t = E_FT.PUMP THEN
	nCheckingTime := GVL_HMI.i_nPumpFeedbackCheckingTime;
ELSE
	nCheckingTime := GVL_HMI.i_nCylinderFeedbackCheckingTime;
END_IF

IF NOT bRising THEN bFeedback := NOT bFeedback; END_IF

IF NOT bFeedback AND NOT FeedbackTimer.IN THEN
    FeedbackTimer(IN := TRUE, PT := INT_TO_TIME(nCheckingTime));	// T#3S
ELSE
	IF bFeedback THEN
		CASE t OF
			E_FT.PUMP:
				IF bRising THEN GVL_HMI.i_nPumpState := 2; ELSE GVL_HMI.i_nPumpState := 4; END_IF
			E_FT.CYL1_E:
				IF bRising THEN GVL_HMI.i_nCylinder1State := 2; END_IF
			E_FT.CYL1_R:
				IF bRising THEN GVL_HMI.i_nCylinder1State := 4; END_IF
			E_FT.CYL2_E:
				IF bRising THEN GVL_HMI.i_nCylinder2State := 2; END_IF
			E_FT.CYL2_R:
				IF bRising THEN GVL_HMI.i_nCylinder2State := 4; END_IF
			E_FT.CYL3_E:
				IF bRising THEN GVL_HMI.i_nCylinder3State := 2; END_IF
			E_FT.CYL3_R:
				IF bRising THEN GVL_HMI.i_nCylinder3State := 4; END_IF
			E_FT.CYL4_E:
				IF bRising THEN GVL_HMI.i_nCylinder4State := 2; END_IF
			E_FT.CYL4_R:
				IF bRising THEN GVL_HMI.i_nCylinder4State := 4; END_IF
			E_FT.CYL5_E:
				IF bRising THEN GVL_HMI.i_nCylinder5State := 2; END_IF
			E_FT.CYL5_R:
				IF bRising THEN GVL_HMI.i_nCylinder5State := 4; END_IF
			E_FT.CYL6_E:
				IF bRising THEN GVL_HMI.i_nCylinder6State := 2; END_IF
			E_FT.CYL6_R:
				IF bRising THEN GVL_HMI.i_nCylinder6State := 4; END_IF
			E_FT.CYL7_E:
				IF bRising THEN GVL_HMI.i_nCylinder7State := 2; END_IF
			E_FT.CYL7_R:
				IF bRising THEN GVL_HMI.i_nCylinder7State := 4; END_IF
			E_FT.PCYL1_E:
				IF bRising THEN GVL_HMI.i_nPCylinder1State := 2; END_IF
			E_FT.PCYL1_R:
				IF bRising THEN GVL_HMI.i_nPCylinder1State := 4; END_IF
			E_FT.PCYL2_E:
				IF bRising THEN GVL_HMI.i_nPCylinder2State := 2; END_IF
			E_FT.PCYL2_R:
				IF bRising THEN GVL_HMI.i_nPCylinder2State := 4; END_IF
		END_CASE
		FeedbackTimer(IN := FALSE);
		o_nResult := 1;
    ELSIF FeedbackTimer.Q THEN
		CASE t OF
			E_FT.PUMP:
				GVL_HMI.i_nPumpState := -1;
				sAlarmMessage := GVL_AlarmMessage.PUMP;
				IF bRising THEN sAlarmMessage := GVL_AlarmMessage.PUMP; ELSE sAlarmMessage := GVL_AlarmMessage.PUMP_OFF; END_IF
			E_FT.CYL1_E:
				GVL_HMI.i_nCylinder1State := -1;
				IF bRising THEN sAlarmMessage := GVL_AlarmMessage.CYL1_NOT_EXTENDED; ELSE sAlarmMessage := GVL_AlarmMessage.CYL1_NOT_EXTENDED_OFF; END_IF
			E_FT.CYL1_R:
				GVL_HMI.i_nCylinder1State := -3;
				IF bRising THEN sAlarmMessage := GVL_AlarmMessage.CYL1_NOT_RETRACTED; ELSE sAlarmMessage := GVL_AlarmMessage.CYL1_NOT_RETRACTED_OFF; END_IF
			E_FT.CYL2_E:
				GVL_HMI.i_nCylinder2State := -1;
				IF bRising THEN sAlarmMessage := GVL_AlarmMessage.CYL2_NOT_EXTENDED; ELSE sAlarmMessage := GVL_AlarmMessage.CYL2_NOT_EXTENDED_OFF; END_IF
			E_FT.CYL2_R:
				GVL_HMI.i_nCylinder2State := -3;
				IF bRising THEN sAlarmMessage := GVL_AlarmMessage.CYL2_NOT_RETRACTED; ELSE sAlarmMessage := GVL_AlarmMessage.CYL2_NOT_RETRACTED_OFF; END_IF
			E_FT.CYL3_E:
				GVL_HMI.i_nCylinder3State := -1;
				IF bRising THEN sAlarmMessage := GVL_AlarmMessage.CYL3_NOT_EXTENDED; ELSE sAlarmMessage := GVL_AlarmMessage.CYL3_NOT_EXTENDED_OFF; END_IF
			E_FT.CYL3_R:
				GVL_HMI.i_nCylinder3State := -3;
				IF bRising THEN sAlarmMessage := GVL_AlarmMessage.CYL3_NOT_RETRACTED; ELSE sAlarmMessage := GVL_AlarmMessage.CYL3_NOT_RETRACTED_OFF; END_IF
			E_FT.CYL4_E:
				GVL_HMI.i_nCylinder4State := -1;
				IF bRising THEN sAlarmMessage := GVL_AlarmMessage.CYL4_NOT_EXTENDED; ELSE sAlarmMessage := GVL_AlarmMessage.CYL4_NOT_EXTENDED_OFF; END_IF
			E_FT.CYL4_R:
				GVL_HMI.i_nCylinder4State := -3;
				IF bRising THEN sAlarmMessage := GVL_AlarmMessage.CYL4_NOT_RETRACTED; ELSE sAlarmMessage := GVL_AlarmMessage.CYL4_NOT_RETRACTED_OFF; END_IF
			E_FT.CYL5_E:
				GVL_HMI.i_nCylinder5State := -1;
				IF bRising THEN sAlarmMessage := GVL_AlarmMessage.CYL5_NOT_EXTENDED; ELSE sAlarmMessage := GVL_AlarmMessage.CYL5_NOT_EXTENDED_OFF; END_IF
			E_FT.CYL5_R:
				GVL_HMI.i_nCylinder5State := -3;
				IF bRising THEN sAlarmMessage := GVL_AlarmMessage.CYL5_NOT_RETRACTED; ELSE sAlarmMessage := GVL_AlarmMessage.CYL5_NOT_RETRACTED_OFF; END_IF
			E_FT.CYL6_E:
				GVL_HMI.i_nCylinder6State := -1;
				IF bRising THEN sAlarmMessage := GVL_AlarmMessage.CYL6_NOT_EXTENDED; ELSE sAlarmMessage := GVL_AlarmMessage.CYL6_NOT_EXTENDED_OFF; END_IF
			E_FT.CYL6_R:
				GVL_HMI.i_nCylinder6State := -3;
				IF bRising THEN sAlarmMessage := GVL_AlarmMessage.CYL6_NOT_RETRACTED; ELSE sAlarmMessage := GVL_AlarmMessage.CYL6_NOT_RETRACTED_OFF; END_IF
			E_FT.CYL7_E:
				GVL_HMI.i_nCylinder7State := -1;
				IF bRising THEN sAlarmMessage := GVL_AlarmMessage.CYL7_NOT_EXTENDED; ELSE sAlarmMessage := GVL_AlarmMessage.CYL7_NOT_EXTENDED_OFF; END_IF
			E_FT.CYL7_R:
				GVL_HMI.i_nCylinder7State := -3;
				IF bRising THEN sAlarmMessage := GVL_AlarmMessage.CYL7_NOT_RETRACTED; ELSE sAlarmMessage := GVL_AlarmMessage.CYL7_NOT_RETRACTED_OFF; END_IF
			E_FT.PCYL1_E:
				GVL_HMI.i_nPCylinder1State := -1;
				IF bRising THEN sAlarmMessage := GVL_AlarmMessage.PCYL1_NOT_EXTENDED; ELSE sAlarmMessage := GVL_AlarmMessage.PCYL1_NOT_EXTENDED_OFF; END_IF
			E_FT.PCYL1_R:
				GVL_HMI.i_nPCylinder1State := -3;
				IF bRising THEN sAlarmMessage := GVL_AlarmMessage.PCYL1_NOT_RETRACTED; ELSE sAlarmMessage := GVL_AlarmMessage.PCYL1_NOT_RETRACTED_OFF; END_IF
			E_FT.PCYL2_E:
				GVL_HMI.i_nPCylinder2State := -1;
				IF bRising THEN sAlarmMessage := GVL_AlarmMessage.PCYL2_NOT_EXTENDED; ELSE sAlarmMessage := GVL_AlarmMessage.PCYL2_NOT_EXTENDED_OFF; END_IF
			E_FT.PCYL2_R:
				GVL_HMI.i_nPCylinder2State := -3;
				IF bRising THEN sAlarmMessage := GVL_AlarmMessage.PCYL2_NOT_RETRACTED; ELSE sAlarmMessage := GVL_AlarmMessage.PCYL2_NOT_RETRACTED_OFF; END_IF
		END_CASE
		
		fSetAlarm( sMsg := sAlarmMessage );
		o_nResult := -1;
    END_IF
END_IF

END_FUNCTION_BLOCK

// ---- POUs/FB_OilPump.TcPOU
FUNCTION_BLOCK FB_OilPump
VAR_INPUT
	i_bCallForCyl: BOOL := TRUE;
END_VAR
VAR_OUTPUT
END_VAR
VAR
    iState : INT := 0;
	FeedbackTimer : TON;
    DelayTimer : TON;
	fSetAlarm : FB_SetAlarm;
	fCheckFeedback : FB_CheckFeedback;
END_VAR

IF GVL_HMI.i_nCmd_Reset = 2 THEN
	IF 20 <= iState AND iState <= 29 THEN
		iState := 0;
	END_IF 
END_IF

CASE iState OF
    0: (* Pump Off, Not Enabled *)
        iState := 10;

    10: (* Pump Enabled from Other Routine *)
		IF GVL_IO.DI_M1 THEN
			DelayAndAdvance( GVL_InitialSetting.PUMP_FAN_DelayTime, iState+1 );
		END_IF
	11:
		GVL_IO.DO_M2 := TRUE;
	    (* Inhibit Pump if DI1.4 or DI1.5 goes Low *)
        IF (NOT GVL_IO.DI_LS1) OR (NOT GVL_IO.DI_TS1) THEN
			GVL_IO.DO_M1 := FALSE;
			GVL_IO.DO_M2 := FALSE;
            iState := iState + 1;
        END_IF
	12: // check to off pump
		IF NOT GVL_IO.DI_M1 THEN
			fCheckFeedback( t := E_FT.PUMP, FeedbackTimer := FeedbackTimer );
		ELSE
			iState := (iState + 10) / 10 * 10;
        END_IF

    20: (* Fault Handling: Check DI1.3 Feedback *)
        (* Start 3-second timer to check for DI1.3 feedback *)
        DelayAndAdvance( GVL_InitialSetting.PUMP_RestartingTime, iState+1 );
	21:
        IF NOT GVL_IO.DI_M1 THEN
			GVL_HMI.i_nPumpState := -1;
			fSetAlarm( sMsg:=GVL_AlarmMessage.PUMP );
			iState := iState / 10 * 10;
		ELSE
			iState := (iState + 10) / 10 * 10;
        END_IF
END_CASE

METHOD DelayAndAdvance : BOOL
VAR_INPUT
	i_nDelayTime: INT;	// ms
	i_nNextState: INT;
END_VAR

VAR
END_VAR
IF NOT DelayTimer.IN THEN
    DelayTimer(IN := TRUE, PT := INT_TO_TIME(i_nDelayTime));
ELSE
    IF DelayTimer.Q THEN 
        iState := i_nNextState; 
    END_IF
END_IF
END_METHOD

END_FUNCTION_BLOCK

// ---- POUs/FB_CorePress.TcPOU
FUNCTION_BLOCK FB_CorePress
VAR_INPUT
END_VAR
VAR_OUTPUT
END_VAR

VAR
    iState : INT := 0;
	FeedbackTimer : TON;
	FeedbackTimerForPCyl : TON;
    DelayTimer : TON;
	fSetAlarm : FB_SetAlarm;
	fCheckFeedback : FB_CheckFeedback;
END_VAR

IF GVL_HMI.i_nCmd_ClearCount = 2 THEN
	GVL_HMI.nProductCount := 0;
END_IF

CASE iState OF
	0: (* Idle/Off, DI_ECS=FALSE *)
		iState := 10;
		
	10: (* check safety conditions *)
		IF GVL_HMI.bSafeties AND GVL_IO.DI_EPD THEN (* Safeties OK and Enable Switch On *)
            GVL_IO.DO_M1 := TRUE; (* Start Oil Pump *)
			CheckFeedback( E_FT.PUMP, TRUE );
			IF GVL_IO.DI_M1 THEN
				DelayAndAdvance(GVL_InitialSetting.PUMP_RunningDelayTime, iState+10);
			END_IF
        END_IF
		
    20: (* Check PCYL1 Retracted, Energize DO6.7 if needed *)
        IF NOT GVL_IO.DI_PCYL1_R THEN
            GVL_IO.DO_PCYL1_R := TRUE; (* Retract PCYL1 *)
			CheckFeedbackForPCyl( E_FT.PCYL1_R, TRUE );
        ELSE
            iState := iState + 10;
        END_IF

    30: (* Count Casing/Core, Move to Next Step When Count Reached *)
        IF (GVL_HMI.nCasingCount >= GVL_HMI.i_nCasingCountForStarting) AND (GVL_HMI.nCoreCount >= GVL_HMI.i_nCoreCountForStarting) THEN
            iState := iState + 10;
        END_IF
		
	40:
        IF NOT GVL_IO.DI_PCYL1_E THEN
            GVL_IO.DO_PCYL1_E := TRUE; (* Extend PCYL1 *)
			CheckFeedback( E_FT.PCYL1_E, TRUE );
        ELSE
			DelayAndAdvance( GVL_HMI.i_nPCylinder1ExtendedRunningTime, iState+1);
        END_IF
	41:
		IF GVL_IO.DI_PCYL1_E THEN
			GVL_IO.DO_PCYL1_E := FALSE;
			CheckFeedback( E_FT.PCYL1_E, FALSE );
		ELSE
			iState := iState + 1;
		END_IF
	42:
        IF NOT GVL_IO.DI_CYL3_E THEN
            GVL_IO.DO_CYL3_E := TRUE; (* Extend CYL3 *)
			CheckFeedback( E_FT.CYL3_E, TRUE );
        ELSE
			DelayAndAdvance( GVL_HMI.i_nCylinder3ExtendedRunningTime, iState+1);
        END_IF
	43:
		IF GVL_IO.DI_CYL3_E THEN
			GVL_IO.DO_CYL3_E := FALSE;
			CheckFeedback( E_FT.CYL3_E, FALSE );
		ELSE
			iState := iState + 1;
		END_IF
	44:
        IF NOT GVL_IO.DI_CYL1_E THEN
            GVL_IO.DO_CYL1_E := TRUE; (* Extend CYL3 *)
			CheckFeedback( E_FT.CYL1_E, TRUE );
        ELSE
			DelayAndAdvance( GVL_HMI.i_nCylinder3ExtendedRunningTime, iState+1);
        END_IF
	45:
		IF GVL_IO.DI_CYL1_E THEN
			GVL_IO.DO_CYL1_E := FALSE;
			CheckFeedback( E_FT.CYL1_E, FALSE );
		ELSE
			iState := (iState + 10) / 10 * 10;
		END_IF
	
	50:
        IF NOT GVL_IO.DI_PCYL1_R THEN
            GVL_IO.DO_PCYL1_R := TRUE;
			CheckFeedback( E_FT.PCYL1_R, TRUE );
        ELSE
			DelayAndAdvance( GVL_HMI.i_nPCylinder1RetractedRunningTime, iState+1);
        END_IF
	51:
		IF GVL_IO.DI_PCYL1_R THEN
			GVL_IO.DO_PCYL1_R := FALSE;
			CheckFeedback( E_FT.PCYL1_R, FALSE );
		ELSE
			iState := iState + 1;
		END_IF
	52:
        IF NOT GVL_IO.DI_CYL3_R THEN
            GVL_IO.DO_CYL3_R := TRUE;
			CheckFeedback( E_FT.CYL3_R, TRUE );
        ELSE
			DelayAndAdvance( GVL_HMI.i_nCylinder3RetractedRunningTime, iState+1);
        END_IF
	53:
		IF GVL_IO.DI_CYL3_R THEN
			GVL_IO.DO_CYL3_R := FALSE;
			CheckFeedback( E_FT.CYL3_R, FALSE );
		ELSE
			iState := iState + 1;
		END_IF
	54:
        IF NOT GVL_IO.DI_CYL1_R THEN
            GVL_IO.DO_CYL1_R := TRUE;
			CheckFeedback( E_FT.CYL1_R, TRUE );
        ELSE
			DelayAndAdvance( GVL_HMI.i_nCylinder1RetractedRunningTime, iState + 1);
        END_IF
	55:
		IF GVL_IO.DI_CYL1_R THEN
			GVL_IO.DO_CYL1_R := FALSE;
			CheckFeedback( E_FT.CYL1_R, FALSE );
		ELSE
			iState := (iState + 10) / 10 * 10;
		END_IF

	60:
        IF NOT GVL_IO.DI_PCYL2_E THEN
            GVL_IO.DO_PCYL2_E := TRUE;
			CheckFeedbackForPCyl( E_FT.PCYL2_E, TRUE );
        ELSE
			DelayAndAdvance( GVL_HMI.i_nPCylinder2ExtendedRunningTime, iState + 10);
        END_IF
		
	70:
        IF NOT GVL_IO.DI_CYL4_E THEN
            GVL_IO.DO_CYL4_E := TRUE;
			CheckFeedback( E_FT.CYL4_E, TRUE );
        ELSE
			DelayAndAdvance( GVL_HMI.i_nCylinder4ExtendedRunningTime, iState+1);
        END_IF
	71:
		IF GVL_IO.DI_CYL4_E THEN
			GVL_IO.DO_CYL4_E := FALSE;
			CheckFeedback( E_FT.CYL4_E, FALSE );
		ELSE
			iState := iState + 1;
		END_IF
	72:
        IF NOT GVL_IO.DI_CYL2_E THEN
            GVL_IO.DO_CYL2_E := TRUE;
			CheckFeedback( E_FT.CYL2_E, TRUE );
        ELSE
			DelayAndAdvance( GVL_HMI.i_nCylinder2ExtendedRunningTime, iState+1);
        END_IF
	73:
		IF GVL_IO.DI_CYL2_E THEN
			GVL_IO.DO_CYL2_E := FALSE;
			CheckFeedback( E_FT.CYL2_E, FALSE );
		ELSE
			iState := (iState + 10) / 10 * 10;
		END_IF
		
	80:
        IF NOT GVL_IO.DI_CYL4_R THEN
            GVL_IO.DO_CYL4_R := TRUE;
			CheckFeedback( E_FT.CYL4_R, TRUE );
        ELSE
			DelayAndAdvance( GVL_HMI.i_nCylinder4RetractedRunningTime, iState+1);
        END_IF
	81:
		IF GVL_IO.DI_CYL4_R THEN
			GVL_IO.DO_CYL4_R := FALSE;
			CheckFeedback( E_FT.CYL4_R, FALSE );
		ELSE
			iState := iState + 1;
		END_IF
	82:
        IF NOT GVL_IO.DI_CYL2_R THEN
            GVL_IO.DO_CYL2_R := TRUE;
			CheckFeedback( E_FT.CYL2_R, TRUE );
        ELSE
			DelayAndAdvance( GVL_HMI.i_nCylinder2RetractedRunningTime, iState+1);
        END_IF
	83:
		IF GVL_IO.DI_CYL2_R THEN
			GVL_IO.DO_CYL2_R := FALSE;
			CheckFeedback( E_FT.CYL2_R, FALSE );
		ELSE
			iState := (iState + 10) / 10 * 10;
		END_IF
	
	90:
		iState := iState + 10;
		
	100:
		iState := iState + 10;

    110: (* Increment product count and loop back to step 2 *)
        GVL_HMI.nProductCount := GVL_HMI.nProductCount + 1;
        iState := 20;
END_CASE

IF 30 < iState AND iState <= 49 THEN
	IF NOT GVL_IO.DI_PCYL1_R THEN
		GVL_IO.DO_PCYL1_R := TRUE; (* Retract PCYL1 *)
		CheckFeedbackForPCyl( E_FT.PCYL1_R, TRUE );
	END_IF
ELSIF 60 < iState AND iState <= 89 THEN
	IF NOT GVL_IO.DI_PCYL2_E THEN
		GVL_IO.DO_PCYL2_E := TRUE;
		CheckFeedbackForPCyl( E_FT.PCYL2_E, TRUE );
	END_IF
END_IF

METHOD CheckFeedback : BOOL
VAR_INPUT
	t : E_FT;
	bRising : BOOL := TRUE;
END_VAR
VAR_OUTPUT
	o_nResult : INT := 0;	// -1: fail, 0: checking, 1: success 
END_VAR
fCheckFeedback(t:=t, bRising:=bRising, FeedbackTimer:=FeedbackTimer);
o_nResult := fCheckFeedback.o_nResult;
END_METHOD

METHOD CheckFeedbackForPCyl : BOOL
VAR_INPUT
	t : E_FT;
	bRising : BOOL := TRUE;
END_VAR
VAR_OUTPUT
	o_nResult : INT := 0;	// -1: fail, 0: checking, 1: success 
END_VAR
fCheckFeedback(t:=t, bRising:=bRising, FeedbackTimer:=FeedbackTimerForPCyl);
o_nResult := fCheckFeedback.o_nResult;
END_METHOD

METHOD DelayAndAdvance : BOOL
VAR_INPUT
	i_nDelayTime: INT;	// ms
	i_nNextState: INT;
END_VAR

VAR
END_VAR
IF NOT DelayTimer.IN THEN
    DelayTimer(IN := TRUE, PT := INT_TO_TIME(i_nDelayTime));
ELSE
    IF DelayTimer.Q THEN 
        iState := i_nNextState; 
    END_IF
END_IF
END_METHOD

END_FUNCTION_BLOCK

// ---- POUs/FB_CasingVibratoryBowl1.TcPOU
FUNCTION_BLOCK FB_CasingVibratoryBowl1
VAR_INPUT
END_VAR
VAR_OUTPUT
END_VAR
VAR
    iState : INT := 0;
    iState2 : INT := 0;
	FeedbackTimer : TON;
    DelayTimer : TON;
	DelayTimer2 : TON;
END_VAR

IF GVL_HMI.i_nCmd_ClearCount = 2 THEN
	GVL_HMI.nCasingCount := 0;
END_IF

CASE iState OF
    0: (* Idle/Off *)
		iState := 10;
	
	10:
        IF GVL_HMI.bSafeties AND GVL_IO.DI_ECS THEN
            iState := iState + 10;
        END_IF

    20: (* Wait for Product in Position *)
		DelayAndAdvance( GVL_InitialSetting.BOWL_RunningDelayTime, iState+1 );
	21:
	    IF GVL_IO.DI_PE1 THEN
            iState := (iState + 10) / 10 * 10;
        END_IF

    30: (* Energize Track Index Solenoid *)
        GVL_IO.DO_PCYL3_E := TRUE;
		DelayAndAdvance( GVL_HMI.i_nPCylinder3ExtendedRunningTime, iState+1 );
	31:
		GVL_IO.DO_PCYL3_E := FALSE;
		iState2 := 0;
        iState := (iState + 10) / 10 * 10;
		
	40:
		DelayAndAdvance( GVL_InitialSetting.PE2_CheckingDelayTime, iState+1 );
	41: (* Check Invert PE and Decide Path *)
		IF GVL_IO.DI_PE2 THEN
			iState := iState + 10;
			DelayTimer.IN := FALSE;
		ELSE
			DelayAndAdvance( GVL_InitialSetting.PE2_MaintainTime, iState+20 );
		END_IF
	
	50:
		GVL_IO.DO_PCYL5_E := TRUE;
		DelayAndAdvance( GVL_HMI.i_nPCylinder5ExtendedRunningTime, iState+1);
	51:
		GVL_IO.DO_PCYL5_E := FALSE;
		GVL_HMI.nCasingCount := GVL_HMI.nCasingCount + 1;
		iState := 20;
		
	60:
		GVL_IO.DO_PCYL4_E := TRUE;
		DelayAndAdvance( GVL_HMI.i_nPCylinder4ExtendedRunningTime, iState+1);
	61:
		GVL_IO.DO_PCYL4_E := FALSE;
		GVL_HMI.nCasingCount := GVL_HMI.nCasingCount + 1;
		iState := (iState + 10) / 10 * 10;
		
	70: (* Check High-Level Sensor *)
		IF GVL_IO.DI_PE4 THEN
			DelayAndAdvance( GVL_HMI.i_nPE4MaintainTime, iState+10 );
		ELSE
			iState := 20;
			DelayTimer.IN := FALSE;
		END_IF
	
	80:
		(* Pause and Wait *)
END_CASE

IF iState >= 20 THEN
	CASE iState2 OF
		0:
			GVL_IO.DO_VB1 := TRUE; 
			IF NOT DelayTimer2.IN THEN
				DelayTimer2(IN := TRUE, PT := INT_TO_TIME(GVL_InitialSetting.VB1_MaintainTime));
			ELSE
				IF DelayTimer2.Q THEN 
					iState2 := iState2 + 10;
				END_IF
			END_IF
		10:
			IF GVL_IO.DI_PE1 THEN
				iState2 := iState2 + 10;
			END_IF
		20:
			(* Stop and Wait *)
	END_CASE
ELSE
	iState2 := 0;
END_IF

METHOD DelayAndAdvance : BOOL
VAR_INPUT
	i_nDelayTime: INT;	// ms
	i_nNextState: INT;
END_VAR

VAR
END_VAR
IF NOT DelayTimer.IN THEN
    DelayTimer(IN := TRUE, PT := INT_TO_TIME(i_nDelayTime));
ELSE
    IF DelayTimer.Q THEN 
        iState := i_nNextState; 
    END_IF
END_IF
END_METHOD

END_FUNCTION_BLOCK

// ---- POUs/FB_CoreVibratoryBowl2.TcPOU
FUNCTION_BLOCK FB_CoreVibratoryBowl2
VAR
    iState : INT := 0;
    iState2 : INT := 0;
	FeedbackTimer : TON;
    DelayTimer : TON;
	DelayTimer2 : TON;
END_VAR

IF GVL_HMI.i_nCmd_ClearCount = 2 THEN
	GVL_HMI.nCoreCount := 0;
END_IF

CASE iState OF
    0: (* Idle/Off *)
		iState := 10;
	
	10:
        IF GVL_HMI.bSafeties AND GVL_IO.DI_ECS THEN
            iState := iState + 10;
        END_IF

    20: (* Wait for Product in Position *)
		DelayAndAdvance( GVL_InitialSetting.BOWL_RunningDelayTime, iState+1 );
	21:
	    IF GVL_IO.DI_PE3 THEN
            iState := (iState + 10) / 10 * 10;
        END_IF

    30: (* Energize Track Index Solenoid *)
        GVL_IO.DO_PCYL6_E := TRUE;
		DelayAndAdvance( GVL_HMI.i_nPCylinder6ExtendedRunningTime, iState+1 );
	31:
		GVL_IO.DO_PCYL3_E := FALSE;
		iState2 := 0;
		GVL_HMI.i_nCoreCountForStarting := GVL_HMI.i_nCoreCountForStarting + 1;
        iState := (iState + 10) / 10 * 10;
		
	40: (* Check High-Level Sensor *)
		IF GVL_IO.DI_PE6 THEN
			DelayAndAdvance( GVL_HMI.i_nPE6MaintainTime, iState+10 );
		ELSE
			iState := 20;
			DelayTimer.IN := FALSE;
		END_IF
	
	80:
		(* Pause and Wait *)
END_CASE

IF iState >= 20 THEN
	CASE iState2 OF
		0:
			GVL_IO.DO_VB2 := TRUE; 
			IF NOT DelayTimer2.IN THEN
				DelayTimer2(IN := TRUE, PT := INT_TO_TIME(GVL_InitialSetting.VB2_MaintainTime));
			ELSE
				IF DelayTimer2.Q THEN 
					iState2 := iState2 + 10;
				END_IF
			END_IF
		10:
			IF GVL_IO.DI_PE3 THEN
				iState2 := iState2 + 10;
			END_IF
		20:
			(* Stop and Wait *)
	END_CASE
ELSE
	iState2 := 0;
END_IF

METHOD DelayAndAdvance : BOOL
VAR_INPUT
	i_nDelayTime: INT;	// ms
	i_nNextState: INT;
END_VAR

VAR
END_VAR
IF NOT DelayTimer.IN THEN
    DelayTimer(IN := TRUE, PT := INT_TO_TIME(i_nDelayTime));
ELSE
    IF DelayTimer.Q THEN 
        iState := i_nNextState; 
    END_IF
END_IF
END_METHOD

END_FUNCTION_BLOCK

// ---- POUs/BaseFuntion/FB_TransmitStatesToHMI.TcPOU
FUNCTION_BLOCK FB_TransmitStatesToHMI
VAR_INPUT
END_VAR
VAR_OUTPUT
END_VAR
VAR
	fSetAlarm : FB_SetAlarm;
END_VAR

// safeties
GVL_HMI.i_b24VDC_CB_OK := GVL_IO.DI_24VDC_CB_OK;
GVL_HMI.i_bESR1 := GVL_IO.DI_ESR1;
GVL_HMI.i_bLS1 := GVL_IO.DI_LS1;
GVL_HMI.i_bTS1 := GVL_IO.DI_TS1;
GVL_HMI.i_bPS1 := GVL_IO.DI_PS1;

// Output
GVL_HMI.i_bVB1 := GVL_IO.DO_VB1;
GVL_HMI.i_bVB2 := GVL_IO.DO_VB2;
GVL_HMI.i_bCyl1E := GVL_IO.DO_CYL1_E;
GVL_HMI.i_bCyl1R := GVL_IO.DO_CYL1_R;
GVL_HMI.i_bCyl2E := GVL_IO.DO_CYL2_E;
GVL_HMI.i_bCyl2R := GVL_IO.DO_CYL2_R;
GVL_HMI.i_bCyl3E := GVL_IO.DO_CYL3_E;
GVL_HMI.i_bCyl3R := GVL_IO.DO_CYL3_R;
GVL_HMI.i_bCyl4E := GVL_IO.DO_CYL4_E;
GVL_HMI.i_bCyl4R := GVL_IO.DO_CYL4_R;
GVL_HMI.i_bCyl5E := GVL_IO.DO_CYL5_E;
GVL_HMI.i_bCyl5R := GVL_IO.DO_CYL5_R;
GVL_HMI.i_bCyl6E := GVL_IO.DO_CYL6_E;
GVL_HMI.i_bCyl6R := GVL_IO.DO_CYL6_R;
GVL_HMI.i_bCyl7E := GVL_IO.DO_CYL7_E;
GVL_HMI.i_bCyl7R := GVL_IO.DO_CYL7_R;
GVL_HMI.i_bCyl8E := GVL_IO.DO_CYL8_E;
GVL_HMI.i_bCyl8R := GVL_IO.DO_CYL8_R;

// core swagging
GVL_HMI.i_bECS := GVL_IO.DI_ECS;
GVL_HMI.i_bEPD := GVL_IO.DI_EPD;
GVL_HMI.i_bJLU := GVL_IO.DI_JLU;

// Vibratory
GVL_HMI.i_bPE1 := GVL_IO.DI_PE1;
IF NOT GVL_HMI.i_bPE1 THEN
	fSetAlarm( sMsg := GVL_AlarmMessage.PE1_FAIL );
END_IF
GVL_HMI.i_bPE2 := GVL_IO.DI_PE2;
IF NOT GVL_HMI.i_bPE2 THEN
	fSetAlarm( sMsg := GVL_AlarmMessage.PE2_FAIL );
END_IF
GVL_HMI.i_bPE3 := GVL_IO.DI_PE3;
IF NOT GVL_HMI.i_bPE3 THEN
	fSetAlarm( sMsg := GVL_AlarmMessage.PE3_FAIL );
END_IF
GVL_HMI.i_bPE4 := GVL_IO.DI_PE4;
IF NOT GVL_HMI.i_bPE4 THEN
	fSetAlarm( sMsg := GVL_AlarmMessage.PE4_FAIL );
END_IF
GVL_HMI.i_bPE5 := GVL_IO.DI_PE5;
IF NOT GVL_HMI.i_bPE5 THEN
	fSetAlarm( sMsg := GVL_AlarmMessage.PE5_FAIL );
END_IF

// analog value
GVL_HMI.i_rPT1 := GVL_IO.AI_PT1;
GVL_HMI.i_rPT2 := GVL_IO.AI_PT2;

// led
IF NOT GVL_HMI.o_bAlarmActive THEN
	GVL_IO.DO_LGreen := FALSE;
	GVL_IO.DO_LRed := TRUE;
ELSE
	GVL_IO.DO_LGreen := TRUE;
	GVL_IO.DO_LRed := FALSE;
END_IF

END_FUNCTION_BLOCK

// ---- POUs/FB_Motor1.TcPOU
FUNCTION_BLOCK FB_Motor1
VAR_INPUT
	new: BOOL;
	pos: REAL;
	vel: REAL;
	acc: REAL;
	dec: REAL;
END_VAR
VAR_OUTPUT
END_VAR
VAR
	will_new: BOOL;
	will_pos: REAL;
	will_vel: REAL;
	will_acc: REAL;
	will_dec: REAL;
	state: E_MoveState;
	PowerAxis: MC_Power;
	PowerAxisOut: ST_McOutputs;
	MoveAxis: MC_MoveAbsolute;
	MoveAbsoluteOut: ST_McOutputs;
	Reset: MC_Reset;
	ResetOut: ST_McOutputs;
END_VAR

GVL_IO.AxisRef1();

IF new THEN
	will_new := TRUE;
	will_pos := pos;
	will_vel := vel;
	will_acc := acc;
	will_dec := dec;
END_IF

CASE state OF
	E_MoveState.init:
		MoveAxis.Execute := FALSE;
		Reset.Execute := FALSE;
		state := E_MoveState.enable;
	E_MoveState.enable:
		PowerAxis.Enable := TRUE;
		PowerAxis.Enable_Positive := TRUE;
		PowerAxis.Enable_Negative := TRUE;
		IF PowerAxis.Status THEN
			state := E_MoveState.forward;
		ELSIF PowerAxis.Error THEN
			state := E_MoveState.error;
		END_IF
	E_MoveState.forward:
		IF will_new THEN
			MoveAxis.Position := will_pos;
			MoveAxis.Velocity := will_vel;
			MoveAxis.Acceleration := will_acc;
			MoveAxis.Deceleration := will_dec;
			MoveAxis.BufferMode := MC_Buffered;
			MoveAxis.Execute := TRUE;
			will_new := FALSE;
		ELSE
			MoveAxis.Execute := FALSE;
		END_IF
		(**IF MoveAxis1.Active THEN
			MoveAxis1.Execute := FALSE;
			state := E_MoveState.new_target_position;
		ELSIF MoveAxis1.CommandAborted OR MoveAxis1.Error THEN
			state := E_MoveState.error;
		END_IF*)
	E_MoveState.error:
		IF GVL_IO.AxisRef1.Status.Error THEN
			state := E_MoveState.reset;
		ELSE
			state := E_MoveState.init;
		END_IF
	E_MoveState.reset:
		Reset.Execute := TRUE;
		IF Reset.Done THEN
			state := E_MoveState.init;
		ELSIF Reset.Error THEN
			state := E_MoveState.init;
		END_IF
END_CASE

ACT_Power();
ACT_Move();
ACT_Reset();

ACTION ACT_Move:
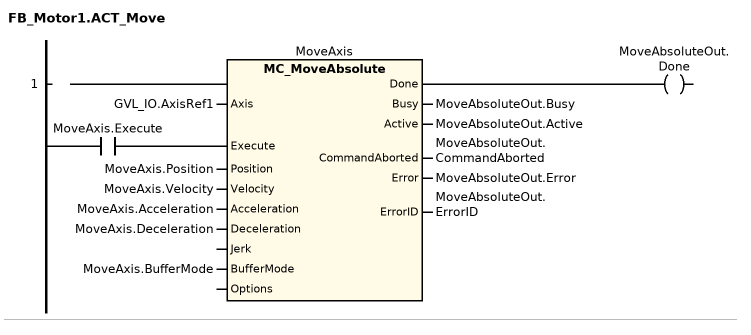
// NETWORK 1
MoveAxis(
    Axis := GVL_IO.AxisRef1,
    Execute := MoveAxis.Execute,
    Position := MoveAxis.Position,
    Velocity := MoveAxis.Velocity,
    Acceleration := MoveAxis.Acceleration,
    Deceleration := MoveAxis.Deceleration,
    BufferMode := MoveAxis.BufferMode,
    Busy => MoveAbsoluteOut.Busy,
    Active => MoveAbsoluteOut.Active,
    CommandAborted => MoveAbsoluteOut.CommandAborted,
    Error => MoveAbsoluteOut.Error,
    ErrorID => MoveAbsoluteOut.ErrorID); // MC_MoveAbsolute
MoveAbsoluteOut.Done := MoveAxis.Done;
END_ACTION

ACTION ACT_Power:
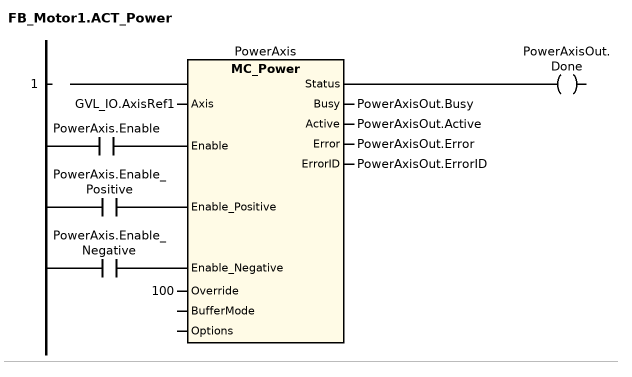
// NETWORK 1
PowerAxis(
    Axis := GVL_IO.AxisRef1,
    Enable := PowerAxis.Enable,
    Enable_Positive := PowerAxis.Enable_Positive,
    Enable_Negative := PowerAxis.Enable_Negative,
    Override := 100,
    Busy => PowerAxisOut.Busy,
    Active => PowerAxisOut.Active,
    Error => PowerAxisOut.Error,
    ErrorID => PowerAxisOut.ErrorID); // MC_Power
PowerAxisOut.Done := PowerAxis.Status;
END_ACTION

ACTION ACT_Reset:
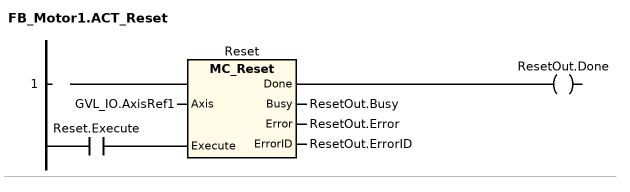
// NETWORK 1
Reset(
    Axis := GVL_IO.AxisRef1,
    Execute := Reset.Execute,
    Busy => ResetOut.Busy,
    Error => ResetOut.Error,
    ErrorID => ResetOut.ErrorID); // MC_Reset
ResetOut.Done := Reset.Done;
END_ACTION

END_FUNCTION_BLOCK
